FUNCTION RandomArrayGenerator : BOOL
VAR_IN_OUT
	aRefArray : ARRAY[1..GVL.nMaximumSizeOfArray] OF REAL;
	nBase : INT;
END_VAR
VAR
	fbRandom : DRAND;
	nIterator : INT;
END_VAR


nBase := nBase + 1;
FOR nIterator  := 1 TO GVL.nMaximumSizeOfArray DO
	fbRandom(seed := nBase + nIterator);
	aRefArray[nIterator] := LREAL_TO_REAL(fbRandom.Num * 700);
END_FOR

END_FUNCTION

(* stored: Version 1.1.0.1, ProductVersion 3.1.4024.16
   POU RandomArrayGenerator: Id {509376b4-9bb7-48b0-8628-60ae4014733d}, SpecialFunc None *)
